(* CODESYS project Spuitinstallatie.project

Project tree, tasks and I/O mapping:
  Device : CODESYS SoftMotion Win V3 64, 3S - Smart Software Solutions GmbH, version 3.5.9.0
    application Application
      libraries: Util, * (System); Standard, * (System)
      task DefaultTask (cyclic, interval T#10ms, priority 16) calls PLC_PRG
      Data types/
      Global Variables/
        global variables Global_Variables
        global variables Variable_Configuration
      POUs/
        program PLC_PRG [IL]
        program visual [ST]
        program Programma_LD [LD]
      Visualizations/
        visualisation Paint_Shop
      trace Sampling_Trace (task ): 
      image pool ImagePool
    SoftMotion General Axis Pool
  GlobalImagePool
  text list GlobalTextList
  text list System
*)

// Device/Application/Global Variables/Global_Variables
VAR_GLOBAL
	Q1: BOOL;
	stop: BOOL;
	start : BOOL;
	Aplus : BOOL;
	Bplus : BOOL;
	Bmin : BOOL;
	Cplus : BOOL;
	Cmin : BOOL;
	a0 : BOOL;
	a1 : BOOL;
	b0 : BOOL;
	b1 : BOOL;
	c0 : BOOL;
	c1 : BOOL;
	Timer_P1 : TON;
	Timer_P2 : TON;
	ET_P1 : TIME;
	ET_P2 : TIME;
	P1 : BOOL;
	P2 : BOOL;
	Teller : CTU;
	antaalPallets : INT;
	d : BOOL;
	reset : BOOL;
	P : BOOL;
	Stock: CTD;
	load: BOOL;
	palletsGedaan: INT;
	palletsVoorraad: INT;
END_VAR

// Device/Application/Global Variables/Variable_Configuration
VAR_CONFIG
END_VAR

// Device/Application/POUs/PLC_PRG
PROGRAM PLC_PRG
VAR
END_VAR

// NETWORK 1
// instruction list
CAL     Programma_LD
CAL     visual

END_PROGRAM

// Device/Application/POUs/Programma_LD
PROGRAM Programma_LD
VAR
END_VAR

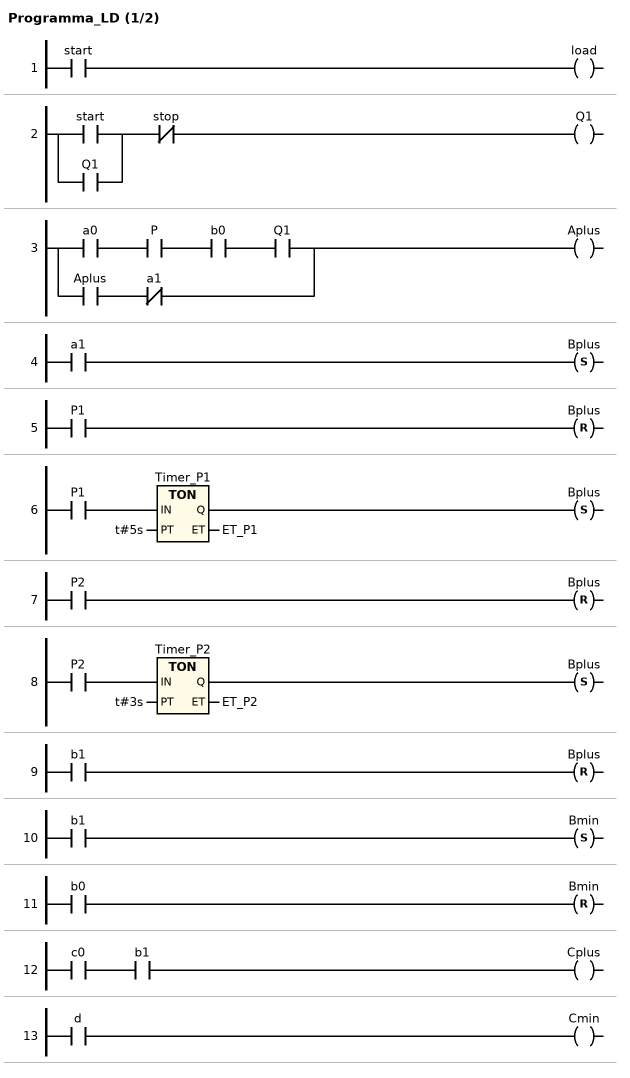
// NETWORK 1
load := start;

// NETWORK 2
Q1 := (start OR Q1) AND NOT stop;

// NETWORK 3
Aplus := a0 AND P AND b0 AND Q1 OR Aplus AND NOT a1;

// NETWORK 4
Bplus S= a1;

// NETWORK 5
Bplus R= P1;

// NETWORK 6
Timer_P1(IN := P1, PT := t#5s, ET => ET_P1); // TON
Bplus S= Timer_P1.Q;

// NETWORK 7
Bplus R= P2;

// NETWORK 8
Timer_P2(IN := P2, PT := t#3s, ET => ET_P2); // TON
Bplus S= Timer_P2.Q;

// NETWORK 9
Bplus R= b1;

// NETWORK 10
Bmin S= b1;

// NETWORK 11
Bmin R= b0;

// NETWORK 12
Cplus := c0 AND b1;

// NETWORK 13
Cmin := d;

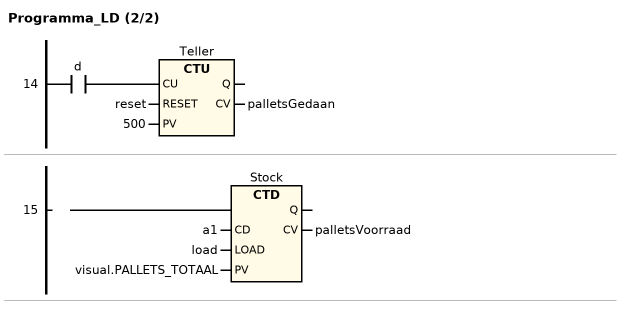
// NETWORK 14
Teller(CU := d, RESET := reset, PV := 500, CV => palletsGedaan); // CTU

// NETWORK 15
Stock(CD := a1, LOAD := load, PV := visual.PALLETS_TOTAAL, CV => palletsVoorraad); // CTD

END_PROGRAM

// Device/Application/POUs/visual
PROGRAM visual
VAR CONSTANT
	ORANJE :INT := 0;
	GEEL :INT := 1;
	BLAUW :INT := 2;
	PALLETS_TOTAAL :INT := 6;
END_VAR
VAR
	(* pallets in de rij van beneden naar boven *)
	palletRij0 : BOOL;
	palletRij1 : BOOL;
	palletRij2 : BOOL;
	palletRij3 : BOOL;
	(* pallet nok de kleur van het pallet *)
	pallet_nok : INT;
	arrayPallets : ARRAY[0..PALLETS_TOTAAL] OF INT := [2,0,1,0,1,2];
	cilinderA: INT;
	cilinderB: INT;
	cilinderC:INT;
	pallet_visual : INT;
	Aplus_visual: BOOL;
	Amin_visual: BOOL;
	Bplus_visual: BOOL;
	Bmin_visual: BOOL;
	Cplus_visual : BOOL;
	Cmin_visual : BOOL;
	terugSlagVanCilinderB: BOOL;
	plusSlagTransportbandD : BOOL;
	spuit_oranje : BOOL;
	spuit_blauw : BOOL;
	spuit_geel : BOOL;
	palletkleur_oranje : BOOL;
	palletkleur_blauw : BOOL;
	palletkleur_geel : BOOL;
	(* tag rotation *)
	tag_blauw : BOOL;
	tag_geel : BOOL;
	tag_oranje : BOOL;
	palletTag_blauw : BOOL;
	palletTag_geel : BOOL;
	palletTag_oranje : BOOL;
	tagging : BOOL;
	i_rotation : INT;
	stempel_blauw : BOOL;
	stempel_oranje : BOOL;
	stempel_geel : BOOL;
	sensor_blauw : BOOL;
	sensor_geel: BOOL;
	sensor_oranje : BOOL;
	terug : BOOL;
END_VAR

(*---------- new programma ---------------*)
(* pallet nok *)
(* nok 0 = oranje , nok 1 = geel, nok 2 = blauw *)
pallet_nok := arrayPallets[Teller.CV];

(* pallet rij *)
IF Q1 AND a0 AND palletsVoorraad = 3 THEN
	palletRij3 := TRUE;
END_IF

IF Q1 AND a0 AND palletsVoorraad = 2 THEN
	palletRij2 := TRUE;
END_IF

IF Q1 AND a0 AND palletsVoorraad = 1 THEN
	palletRij1 := TRUE;
END_IF

IF Q1 AND a0 AND palletsVoorraad = 0 THEN
	palletRij0 := TRUE;
END_IF

IF palletsVoorraad = 0 THEN 
	P := FALSE;
ELSE 
	P := TRUE;
END_IF

(* cilinder A *)
IF Aplus THEN
	IF cilinderA < 150 THEN
		cilinderA := cilinderA + 1;
	END_IF
ELSE
	IF cilinderA > 0 THEN
		cilinderA := cilinderA - 1;
	END_IF
END_IF

CASE cilinderA OF
	  0: a0 := TRUE;
	  5: a0 := FALSE;
	145: a1 := FALSE;
	150: a1 := TRUE;
END_CASE

(* cilinder B *)
IF Bplus THEN
	IF cilinderB < 560 THEN
		cilinderB := cilinderB + 1;
	END_IF
END_IF

IF Bmin THEN
	IF cilinderB > 0 THEN
		cilinderB := cilinderB -1;
	END_IF
END_IF

CASE cilinderB OF
	  0: b0 := TRUE;
	  5: b0 := FALSE;
	555: b1 := FALSE;
	560: b1 := TRUE;
END_CASE

(* stop voor spuitkabine 1 en 2 alleen bij de plus slag *)
CASE cilinderB OF
	180: IF NOT terugSlagVanCilinderB THEN P1 := TRUE; END_IF
	360: IF NOT terugSlagVanCilinderB THEN P2 := TRUE; END_IF
END_CASE

(* nok 0 = oranje , nok 1 = geel, nok 2 = blauw *)
IF cilinderA > 80 AND pallet_nok = 0 THEN
	sensor_oranje := TRUE;
END_IF

IF cilinderA > 80 AND pallet_nok = 1 THEN
	sensor_geel := TRUE;
END_IF

IF cilinderA > 80 AND pallet_nok = 2 THEN
	sensor_blauw := TRUE;
END_IF

(* gaa verder met cilinderB als timer P1 true is *)
IF Timer_P1.Q THEN
	P1 := FALSE;
END_IF

IF Timer_P2.Q THEN
	P2 := FALSE;
END_IF

(* spuitkabine and palletkleur *)
IF pallet_nok = 0 AND P1 THEN
	spuit_oranje := TRUE;
	palletkleur_oranje := TRUE;
ELSE 
	spuit_oranje := FALSE;
END_IF

IF pallet_nok = 1 AND P1 THEN
	spuit_geel := TRUE;
	palletkleur_geel := TRUE;
ELSE
	spuit_geel := FALSE;
END_IF

IF pallet_nok = 2 AND P1 THEN
	spuit_blauw := TRUE;
	palletkleur_blauw := TRUE;
ELSE
	spuit_blauw := FALSE;
END_IF

(* Tagkabine and palletTag *)
IF pallet_nok = 0 AND P2 THEN
	(* P2 till timer ends *)
	tag_oranje := TRUE;
	IF tagging THEN
		(* Tag on pallet till reset sensor d *)
		palletTag_oranje := TRUE;
	END_IF
ELSE 
	tag_oranje := FALSE;
END_IF

IF pallet_nok = 1 AND P2 THEN
	tag_geel := TRUE;
	IF tagging THEN
		(* Tag on pallet till reset sensor d *)
		palletTag_geel := TRUE;
	END_IF
ELSE
	tag_geel := FALSE;
END_IF

IF pallet_nok = 2 AND P2 THEN
	tag_blauw := TRUE;
	IF tagging THEN
		(* Tag on pallet BOOL till reset sensor d *)
		palletTag_blauw := TRUE;
	END_IF
ELSE
	tag_blauw := FALSE;
END_IF

IF i_rotation >= 70 THEN 
	tagging := TRUE;
END_IF

IF i_rotation <= 0 THEN
	tagging := FALSE;
END_IF

(* Tag rotation *)
IF P2 THEN
	IF i_rotation < 70 THEN
		i_rotation := i_rotation + 1; 
	END_IF
ELSE
	IF i_rotation > 0 THEN
		i_rotation := i_rotation - 1;
	END_IF
END_IF

(* nok 0 = oranje , nok 1 = geel, nok 2 = blauw *)
IF i_rotation > 1 AND pallet_nok = 2 THEN
	stempel_blauw := TRUE;
ELSE 
	stempel_blauw := FALSE;
END_IF

IF i_rotation > 1 AND pallet_nok = 0 THEN
	stempel_oranje := TRUE;
ELSE 
	stempel_oranje := FALSE;
END_IF

IF i_rotation > 1 AND pallet_nok = 1 THEN
	stempel_geel := TRUE;
ELSE 
	stempel_geel := FALSE;
END_IF

(* voorkom dat de timer bij het terugslag weer gaat tellen *)
IF b1 THEN
	terugSlagVanCilinderB := TRUE;
END_IF

IF b0 THEN
	terugSlagVanCilinderB := FALSE;
END_IF

(* cilinder C *)
IF Cplus THEN
	Cplus_visual := TRUE;
	Cmin_visual := FALSE;
END_IF

IF Cmin THEN 
	Cmin_visual := TRUE;
	Cplus_visual := FALSE;
END_IF

IF Cplus_visual THEN
	IF cilinderC > - 50 THEN
		cilinderC := cilinderC - 1;
	END_IF
END_IF

IF Cmin_visual THEN
	IF cilinderC < 0 THEN
		cilinderC := cilinderC + 1;
	END_IF
END_IF

CASE cilinderC OF
	  0: c0 := TRUE;
	 -5: c0 := FALSE;
	-45: c1 := FALSE;
	-50: c1 := TRUE; 
END_CASE

(* pallet visualisatie op het einde eindschakelaar d wordt bediend *)
IF c1 THEN
	IF pallet_visual < 140 THEN
		pallet_visual := pallet_visual + 1;
		plusSlagTransportbandD := TRUE;
	END_IF
ELSE
	plusSlagTransportbandD := FALSE;
END_IF

IF pallet_visual = 140 THEN
	d := TRUE;
END_IF 

(* reset palletkleur palletTag and rotation*)
IF d THEN 
	palletkleur_oranje := FALSE;
	palletkleur_blauw := FALSE;
	palletkleur_geel := FALSE;
	palletTag_oranje := FALSE;
	palletTag_blauw := FALSE;
	palletTag_geel := FALSE;
	i_rotation := 0;
	tagging := FALSE;
	sensor_oranje := FALSE;
	sensor_geel := FALSE;
	sensor_blauw := FALSE;
END_IF

(* reset eindschakelaar d en reset pallet_visual loopband *)
IF c0 THEN
	d := FALSE;
	pallet_visual := 0;
END_IF

(*---------------- einde new programma ------------------------------*)

END_PROGRAM

// Device/Application/Visualizations/Paint_Shop
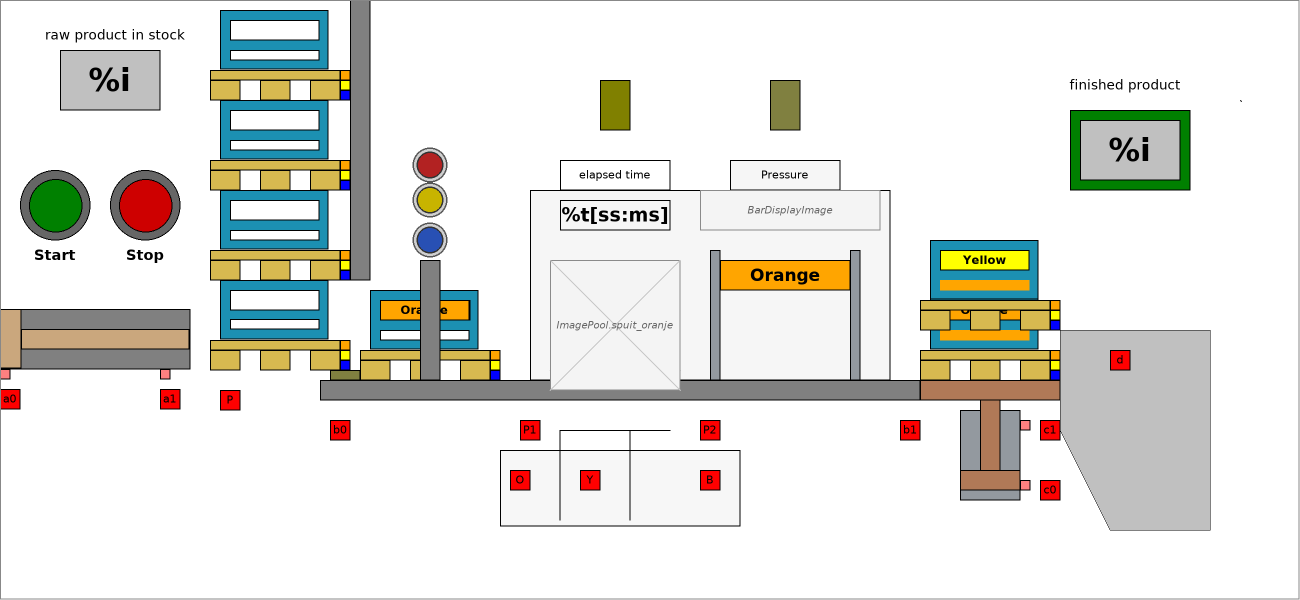
VISUALIZATION Paint_Shop  // 1300x600, background image ImagePool.industrial
    Rectangle (500,450 240x76)
    Polygon (1060,430) (1060,330) (1210,330) (1210,530) (1110,530)
    Rectangle (1070,110 120x80), text variable: Global_Variables.Teller.CV, colour toggle: Global_Variables.d
    Line (630,520) (630,430)
    Line (560,520) (560,430)
    Rectangle (530,190 360x190)
    Polyline (540,210)
    Rectangle (320,380 600x20)
    Rectangle (350,0 20x280)
    Rectangle (560,160 110x30), "elapsed time"
    Rectangle (730,160 110x30), "Pressure"
    Polygon (660,480), colour toggle: visual.spuit_geel
    Polygon (660,460), colour toggle: visual.spuit_geel
    Polygon (690,480), colour toggle: visual.spuit_blauw
    Polygon (690,460), colour toggle: visual.spuit_blauw
    Group (570,250 80x10)
        Polyline (560,220)
        Polyline (590,220)
        Polyline (600,220)
        Polyline (610,220)
        Polyline (620,220)
        Polyline (630,220)
        Polyline (640,220)
    Rectangle (720,260 130x30), invisible if: visual.i_rotation > 1
    Polyline (610,470)
    Polyline (710,470)
    Rectangle (580,470 20x20), "Y", colour toggle: visual.spuit_geel
    Rectangle (700,470 20x20), "B", colour toggle: visual.spuit_blauw
    Polygon (670,160)
    Polygon (840,160)
    RoundedRectangle (600,80 30x50)
    RoundedRectangle (770,80 30x50)
    Rectangle (0,309 190x60)
    Rectangle (0,369 10x10)
    Rectangle (160,369 10x10)
    Rectangle (0,389 20x20), "a0", colour toggle: a0
    Rectangle (160,389 20x20), "a1", colour toggle: a1
    Group (0,280 209x88)
        p3560616238: visual.cilinderA
        Rectangle (21,49 168x20)
        Polygon (190,60)
        Rectangle (0,29 21x59)
    Polygon (350,410)
    Polygon (920,410)
    Rectangle (330,420 20x20), "b0", colour toggle: b0
    Rectangle (900,420 20x20), "b1", colour toggle: Programma_LD.b1
    Polygon (540,410)
    Polygon (720,410)
    Rectangle (520,420 20x20), "P1", colour toggle: P1
    Rectangle (700,420 20x20), "P2", colour toggle: P2
    Rectangle (330,370 30x10)
        p3560616238: visual.cilinderB
    Polygon (210,450)
    Rectangle (960,410 60x90)
    Rectangle (1020,420 10x10)
    Rectangle (1020,480 10x10)
    Rectangle (1040,420 20x20), "c1", colour toggle: c1
    Rectangle (1040,480 20x20), "c0", colour toggle: Global_Variables.c0
    Group (920,380 140x110)
        p2773130477: visual.cilinderC
        p1126004900: visual.cilinderC
        Rectangle (60,10 20x100)
        Rectangle (0,0 140x20)
        Rectangle (40,90 60x20)
    Polygon (920,410)
    Rectangle (1110,350 20x20), "d", colour toggle: d
    Rectangle (1080,120 100x60), "%i", text variable: Global_Variables.palletsGedaan
    Group (210,280 140x90), invisible if: NOT a0 AND NOT Aplus OR visual.palletRij0
        p3560616238: visual.cilinderA
        Rectangle (0,70 30x20)
        Rectangle (100,70 30x20)
        Rectangle (50,70 30x20)
        Rectangle (10,0 108x59)
        Rectangle (20,10 89x20)
        Rectangle (20,39 89x10)
        Rectangle (0,60 130x10)
        Rectangle (130,60 10x10), invisible if: visual.pallet_nok = 1 OR visual.pallet_nok = 2
        Rectangle (130,70 10x10), invisible if: visual.pallet_nok = 0 OR visual.pallet_nok = 2
        Rectangle (130,80 10x10), invisible if: visual.pallet_nok = 0 OR visual.pallet_nok = 1
        Group (0,0 140x90), invisible if: NOT Aplus
            Rectangle (0,70 30x20)
            Rectangle (100,70 30x20)
            Rectangle (50,70 30x20)
            Rectangle (10,0 108x59)
            Rectangle (20,10 89x20)
            Rectangle (20,39 89x10)
            Rectangle (0,60 130x10)
            Rectangle (130,60 10x10), invisible if: visual.pallet_nok = 1 OR visual.pallet_nok = 2
            Rectangle (130,70 10x10), invisible if: visual.pallet_nok = 0 OR visual.pallet_nok = 2
            Rectangle (130,80 10x10), invisible if: visual.pallet_nok = 0 OR visual.pallet_nok = 1
            Group (0,0 140x90), invisible if: Aplus
                Rectangle (0,70 30x20)
                Rectangle (100,70 30x20)
                Rectangle (50,70 30x20)
                Rectangle (10,0 108x59)
                Rectangle (20,10 89x20)
                Rectangle (20,39 89x10)
                Rectangle (0,60 130x10)
                Rectangle (130,60 10x10), invisible if: visual.pallet_nok = 1 OR visual.pallet_nok = 2
                Rectangle (130,70 10x10), invisible if: visual.pallet_nok = 0 OR visual.pallet_nok = 2
                Rectangle (130,80 10x10), invisible if: visual.pallet_nok = 0 OR visual.pallet_nok = 1
                Group (0,0 140x90), invisible if: NOT Aplus
                    Rectangle (0,70 30x20)
                    Rectangle (100,70 30x20)
                    Rectangle (50,70 30x20)
                    Rectangle (10,0 108x59)
                    Rectangle (20,10 89x20)
                    Rectangle (20,39 89x10)
                    Rectangle (0,60 130x10)
                    Rectangle (130,60 10x10), invisible if: visual.pallet_nok = 1 OR visual.pallet_nok = 2
                    Rectangle (130,70 10x10), invisible if: visual.pallet_nok = 0 OR visual.pallet_nok = 2
                    Rectangle (130,80 10x10), invisible if: visual.pallet_nok = 0 OR visual.pallet_nok = 1
    Polygon (350,410)
    Rectangle (220,390 20x20), "P", colour toggle: Global_Variables.P
    Group (210,190 140x90), invisible if: visual.palletRij1
        Rectangle (0,70 30x20)
        Rectangle (100,70 30x20)
        Rectangle (50,70 30x20)
        Rectangle (10,0 108x59)
        Rectangle (20,10 89x20)
        Rectangle (20,39 89x10)
        Rectangle (0,60 130x10)
        Rectangle (130,60 10x10), invisible if: visual.pallet_nok = 1 OR visual.pallet_nok = 2
        Rectangle (130,70 10x10), invisible if: visual.pallet_nok = 0 OR visual.pallet_nok = 2
        Rectangle (130,80 10x10), invisible if: visual.pallet_nok = 0 OR visual.pallet_nok = 1
        Rectangle (0,70 30x20)
        Rectangle (100,70 30x20)
        Rectangle (50,70 30x20)
        Rectangle (10,0 108x59)
        Rectangle (20,10 89x20)
        Rectangle (20,39 89x10)
        Rectangle (0,60 130x10)
        Rectangle (130,60 10x10), invisible if: visual.pallet_nok = 1 OR visual.pallet_nok = 2
        Rectangle (130,70 10x10), invisible if: visual.pallet_nok = 0 OR visual.pallet_nok = 2
        Rectangle (130,80 10x10), invisible if: visual.pallet_nok = 0 OR visual.pallet_nok = 1
        Rectangle (0,70 30x20)
        Rectangle (100,70 30x20)
        Rectangle (50,70 30x20)
        Rectangle (10,0 108x59)
        Rectangle (20,10 89x20)
        Rectangle (20,39 89x10)
        Rectangle (0,60 130x10)
        Rectangle (130,60 10x10), invisible if: visual.pallet_nok = 1 OR visual.pallet_nok = 2
        Rectangle (130,70 10x10), invisible if: visual.pallet_nok = 0 OR visual.pallet_nok = 2
        Rectangle (130,80 10x10), invisible if: visual.pallet_nok = 0 OR visual.pallet_nok = 1
        Rectangle (0,70 30x20)
        Rectangle (100,70 30x20)
        Rectangle (50,70 30x20)
        Rectangle (10,0 108x59)
        Rectangle (20,10 89x20)
        Rectangle (20,40 89x10)
        Rectangle (0,60 130x10)
        Rectangle (130,60 10x10)
        Rectangle (130,70 10x10)
        Rectangle (130,80 10x10)
    Group (920,290 140x90), invisible if: Global_Variables.c0 OR visual.Cmin_visual OR Global_Variables.c1
        p2738717112: visual.cilinderC
        Rectangle (10,0 108x59)
        Rectangle (0,70 30x20)
        Rectangle (100,70 30x20)
        Rectangle (50,70 30x20)
        Rectangle (0,60 130x10)
        Rectangle (130,60 10x10), invisible if: visual.pallet_nok = 1 OR visual.pallet_nok = 2
        Rectangle (130,70 10x10), invisible if: visual.pallet_nok = 0 OR visual.pallet_nok = 2
        Rectangle (130,80 10x10), invisible if: visual.pallet_nok = 0 OR visual.pallet_nok = 1
        Rectangle (20,10 89x20), "Blue", invisible if: NOT visual.palletTag_blauw
        Rectangle (20,10 89x20), "Yellow", invisible if: NOT visual.palletTag_geel
        Rectangle (20,10 89x20), "Orange", invisible if: NOT visual.palletTag_oranje
        Rectangle (20,40 89x10), invisible if: NOT visual.palletkleur_blauw
        Rectangle (20,40 89x10), invisible if: NOT visual.palletkleur_geel
        Rectangle (20,40 89x10), invisible if: NOT visual.palletkleur_oranje
    Group (920,240 140x90), invisible if: NOT visual.plusSlagTransportbandD
        p3560616238: visual.pallet_visual
        Rectangle (0,70 30x20)
        Rectangle (100,70 30x20)
        Rectangle (50,70 30x20)
        Rectangle (10,0 108x59)
        Rectangle (0,60 130x10)
        Rectangle (130,60 10x10), invisible if: visual.pallet_nok = 1 OR visual.pallet_nok = 2
        Rectangle (130,70 10x10), invisible if: visual.pallet_nok = 0 OR visual.pallet_nok = 2
        Rectangle (130,80 10x10), invisible if: visual.pallet_nok = 0 OR visual.pallet_nok = 1
        Rectangle (20,10 89x20), "Orange", invisible if: NOT visual.palletTag_oranje
        Rectangle (20,10 89x20), "Blue", invisible if: NOT visual.palletTag_blauw
        Rectangle (20,10 89x20), "Yellow", invisible if: NOT visual.palletTag_geel
        Rectangle (20,40 89x10), invisible if: NOT visual.palletkleur_blauw
        Rectangle (20,40 89x10), invisible if: NOT visual.palletkleur_geel
        Rectangle (20,40 89x10), invisible if: NOT visual.palletkleur_oranje
    Line (560,430) (670,430)
    Polygon (660,480), colour toggle: visual.spuit_oranje
    Polygon (660,460), colour toggle: visual.spuit_oranje
    Polyline (610,470)
    Rectangle (510,470 20x20), "O", colour toggle: visual.spuit_oranje
    Textfield (560,200 110x30), "%t[ss:ms]", text variable: Timer_P1.ET
    Line (720,90)
    Line (720,380) (720,250)
    Group (360,290 140x90), invisible if: visual.terugSlagVanCilinderB OR Global_Variables.b0
        p3560616238: visual.cilinderB
        Rectangle (10,0 108x59)
        Rectangle (20,10 89x20), "Geel", invisible if: NOT visual.palletTag_geel
        Rectangle (20,10 89x20), "Blauw", invisible if: NOT visual.palletTag_blauw
        Rectangle (20,10 89x20), "Oranje", invisible if: NOT visual.palletTag_oranje
        Rectangle (20,40 89x10), invisible if: NOT visual.palletkleur_oranje
        Rectangle (20,40 89x10), invisible if: NOT visual.palletkleur_geel
        Rectangle (20,40 89x10), invisible if: NOT visual.palletkleur_blauw
        Rectangle (20,40 89x10), invisible if: visual.palletkleur_blauw OR visual.palletkleur_geel OR visual.palletkleur_oranje
        Rectangle (20,10 89x20), invisible if: visual.palletTag_blauw OR visual.palletTag_geel OR visual.palletTag_oranje
        Rectangle (0,70 30x20)
        Rectangle (100,70 30x20)
        Rectangle (50,70 30x20)
        Rectangle (0,60 130x10)
        Rectangle (130,60 10x10), invisible if: visual.pallet_nok = 1 OR visual.pallet_nok = 2
        Rectangle (130,70 10x10), invisible if: visual.pallet_nok = 0 OR visual.pallet_nok = 2
        Rectangle (130,80 10x10), invisible if: visual.pallet_nok = 0 OR visual.pallet_nok = 1
        Rectangle (20,10 89x20), invisible if: NOT visual.palletkleur_blauw
        Rectangle (20,10 90x20), invisible if: NOT visual.palletkleur_geel
        Rectangle (20,10 89x20), invisible if: NOT visual.palletkleur_oranje
        Rectangle (20,10 89x20), "Blue", invisible if: NOT visual.palletTag_blauw
        Rectangle (20,10 90x20), "Yellow", invisible if: NOT visual.palletTag_geel
        Rectangle (20,10 89x20), "Orange", invisible if: NOT visual.palletTag_oranje
    Rectangle (850,250 10x130)
    Rectangle (710,250 10x130)
    Group (210,100 140x90), invisible if: visual.palletRij2
        Rectangle (0,70 30x20)
        Rectangle (100,70 30x20)
        Rectangle (50,70 30x20)
        Rectangle (10,0 108x59)
        Rectangle (20,10 89x20)
        Rectangle (20,39 89x10)
        Rectangle (0,60 130x10)
        Rectangle (130,60 10x10), invisible if: visual.pallet_nok = 1 OR visual.pallet_nok = 2
        Rectangle (130,70 10x10), invisible if: visual.pallet_nok = 0 OR visual.pallet_nok = 2
        Rectangle (130,80 10x10), invisible if: visual.pallet_nok = 0 OR visual.pallet_nok = 1
        Rectangle (0,70 30x20)
        Rectangle (100,70 30x20)
        Rectangle (50,70 30x20)
        Rectangle (10,0 108x59)
        Rectangle (20,10 89x20)
        Rectangle (20,39 89x10)
        Rectangle (0,60 130x10)
        Rectangle (130,60 10x10), invisible if: visual.pallet_nok = 1 OR visual.pallet_nok = 2
        Rectangle (130,70 10x10), invisible if: visual.pallet_nok = 0 OR visual.pallet_nok = 2
        Rectangle (130,80 10x10), invisible if: visual.pallet_nok = 0 OR visual.pallet_nok = 1
        Rectangle (0,70 30x20)
        Rectangle (100,70 30x20)
        Rectangle (50,70 30x20)
        Rectangle (10,0 108x59)
        Rectangle (20,10 89x20)
        Rectangle (20,39 89x10)
        Rectangle (0,60 130x10)
        Rectangle (130,60 10x10), invisible if: visual.pallet_nok = 1 OR visual.pallet_nok = 2
        Rectangle (130,70 10x10), invisible if: visual.pallet_nok = 0 OR visual.pallet_nok = 2
        Rectangle (130,80 10x10), invisible if: visual.pallet_nok = 0 OR visual.pallet_nok = 1
        Rectangle (0,70 30x20)
        Rectangle (100,70 30x20)
        Rectangle (50,70 30x20)
        Rectangle (10,0 108x59)
        Rectangle (20,10 89x20)
        Rectangle (20,40 89x10)
        Rectangle (0,60 130x10)
        Rectangle (130,60 10x10)
        Rectangle (130,70 10x10)
        Rectangle (130,80 10x10)
    Group (210,10 140x90), invisible if: visual.palletRij3
        Rectangle (0,70 30x20)
        Rectangle (100,70 30x20)
        Rectangle (50,70 30x20)
        Rectangle (10,0 108x59)
        Rectangle (20,10 89x20)
        Rectangle (20,39 89x10)
        Rectangle (0,60 130x10)
        Rectangle (130,60 10x10), invisible if: visual.pallet_nok = 1 OR visual.pallet_nok = 2
        Rectangle (130,70 10x10), invisible if: visual.pallet_nok = 0 OR visual.pallet_nok = 2
        Rectangle (130,80 10x10), invisible if: visual.pallet_nok = 0 OR visual.pallet_nok = 1
        Rectangle (0,70 30x20)
        Rectangle (100,70 30x20)
        Rectangle (50,70 30x20)
        Rectangle (10,0 108x59)
        Rectangle (20,10 89x20)
        Rectangle (20,39 89x10)
        Rectangle (0,60 130x10)
        Rectangle (130,60 10x10), invisible if: visual.pallet_nok = 1 OR visual.pallet_nok = 2
        Rectangle (130,70 10x10), invisible if: visual.pallet_nok = 0 OR visual.pallet_nok = 2
        Rectangle (130,80 10x10), invisible if: visual.pallet_nok = 0 OR visual.pallet_nok = 1
        Rectangle (0,70 30x20)
        Rectangle (100,70 30x20)
        Rectangle (50,70 30x20)
        Rectangle (10,0 108x59)
        Rectangle (20,10 89x20)
        Rectangle (20,39 89x10)
        Rectangle (0,60 130x10)
        Rectangle (130,60 10x10), invisible if: visual.pallet_nok = 1 OR visual.pallet_nok = 2
        Rectangle (130,70 10x10), invisible if: visual.pallet_nok = 0 OR visual.pallet_nok = 2
        Rectangle (130,80 10x10), invisible if: visual.pallet_nok = 0 OR visual.pallet_nok = 1
        Rectangle (0,70 30x20)
        Rectangle (100,70 30x20)
        Rectangle (50,70 30x20)
        Rectangle (10,0 108x59)
        Rectangle (20,10 89x20)
        Rectangle (20,40 89x10)
        Rectangle (0,60 130x10)
        Rectangle (130,60 10x10)
        Rectangle (130,70 10x10)
        Rectangle (130,80 10x10)
    Lamp1 (410,180 40x40), variable: visual.sensor_geel, style: Lamp-Lamp1-Yellow
    Lamp1 (410,220 40x40), variable: visual.sensor_blauw, style: Lamp-Lamp1-Blue
    Lamp1 (410,140 40x50), variable: visual.sensor_oranje, style: Lamp-Lamp1-Red
    Rectangle (720,260 130x30), "Yellow", invisible if: NOT visual.stempel_geel
        p2773130477: visual.i_rotation
    Rectangle (720,260 130x30), "Blue", invisible if: NOT visual.stempel_blauw
        p2773130477: visual.i_rotation
    Rectangle (720,260 130x30), "Orange", invisible if: NOT visual.stempel_oranje
        p2773130477: visual.i_rotation
    Rectangle (420,260 20x120)
    Polygon (1240,100) (1241,101)
    Rectangle (60,50 100x60), "%i", text variable: Global_Variables.palletsVoorraad
    Label (40,20 150x30), "raw product in stock"
    Label (1050,70 150x30), "finished product"
    Label (30,240 50x30), "Start"
    Label (120,240 50x30), "Stop"
    BarDisplayImage (700,190 180x40), value: visual.i_rotation, style: BarDisplayImage-Gray, scale format: %.1f, scale 0..70
    Ellipse (20,170 70x70)
    Ellipse (29,179 53x53)
        tap Global_Variables.start
    Ellipse (110,170 70x70)
    Ellipse (119,179 53x53)
    Image (560,260 120x110), invisible if: NOT visual.spuit_blauw, image: ImagePool.spuit_blauw
    Image (550,260 130x110), invisible if: NOT visual.spuit_geel, image: ImagePool.spuit_geel
    Image (550,260 130x130), invisible if: NOT visual.spuit_oranje, image: ImagePool.spuit_oranje
END_VISUALIZATION

(* text list System (id | default)
  Apr | Apr
  April | April
  Aug | Aug
  August | August
  Dec | Dec
  December | December
  Feb | Feb
  February | February
  Fri | Fri
  Friday | Friday
  Jan | Jan
  January | January
  Jul | Jul
  July | July
  Jun | Jun
  June | June
  Mar | Mar
  March | March
  May | May
  May_3Letter | May
  Mon | Mon
  Monday | Monday
  Nov | Nov
  November | November
  Oct | Oct
  October | October
  Sat | Sat
  Saturday | Saturday
  Sep | Sep
  September | September
  Sun | Sun
  Sunday | Sunday
  Thu | Thu
  Thursday | Thursday
  Tue | Tue
  Tuesday | Tuesday
  Wed | Wed
  Wednesday | Wednesday
   |  *)
